GLOBALCONSTANTS bitconst (* Global constants *)
  (* Standard: 61499-1 *)
  (* Version 1.0, 2024-02-22, franz *)
  VAR_GLOBAL CONSTANT
    BOOL_BIT_ZZ : BOOL := 2#0; (* ZERO Constant *)
    BOOL_BIT_00 : BOOL := 2#1; (* Bit 0 Constant *)
    BYTE_BIT_ZZ : BYTE := 2#0000_0000; (* ZERO Constant *)
    BYTE_BIT_00 : BYTE := 2#0000_0001; (* Bit 0 Constant *)
  END_VAR
END_GLOBALCONSTANTS
